Yaskawa INFORM job: neg_x_1.JBI

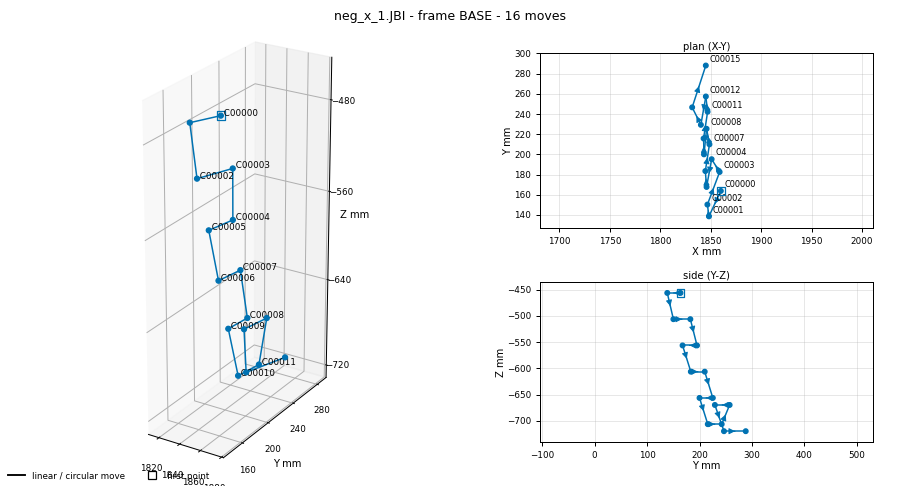
[picture p0: tool path of neg_x_1.JBI in frame BASE, 16 of 18 moves have a stored position in this frame; points joined in program order, loops and branches not executed]
/JOB
//NAME neg_x_1
//POS
///NPOS 16,0,16,0,0,0
///TOOL 0
///POSTYPE BASE
///RECTAN
///RCONF 0,0,0,0,0,0,0,0,0,0,0,0,0,0,0,0,0,0,0,0,0,0,0,0
C00000=1860.009400,163.782870,-456.169200,-175.000000,-80.909620,-24.601701
C00001=1848.219400,138.594450,-456.169200,-175.000000,-80.909620,-24.601701
C00002=1846.699400,150.259350,-506.169200,-175.000000,-80.909620,-24.601701
C00003=1858.829400,182.584150,-506.169200,-175.000000,-80.909620,-24.601701
C00004=1850.899400,195.228650,-556.169200,-175.000000,-80.909620,-24.601701
C00005=1845.879400,167.731640,-556.169200,-175.000000,-80.909620,-24.601701
C00006=1844.649400,183.479050,-606.169200,-175.000000,-80.909620,-24.601701
C00007=1848.749400,209.941950,-606.169200,-175.000000,-80.909620,-24.601701
C00008=1845.889400,225.378650,-656.169200,-175.000000,-80.909620,-24.601701
C00009=1843.319400,200.049150,-656.169200,-175.000000,-80.909620,-24.601701
C00010=1842.919400,215.770950,-706.169200,-175.000000,-80.909620,-24.601701
C00011=1846.899400,242.289250,-706.169200,-175.000000,-80.909620,-24.601701
C00012=1845.159400,257.405150,-669.566660,180.000000,-60.000000,0.000000
C00013=1840.239400,229.288350,-669.566660,180.000000,-60.000000,0.000000
C00014=1831.609400,246.639550,-719.566660,180.000000,-60.000000,0.000000
C00015=1845.119400,288.075850,-719.566660,180.000000,-60.000000,0.000000
///POSTYPE PULSE
///PULSE
EX000=92160
///POSTYPE PULSE
///PULSE
EC00000=92160
EC00001=92160
EC00002=92160
EC00003=92160
EC00004=92160
EC00005=92160
EC00006=92160
EC00007=92160
EC00008=92160
EC00009=92160
EC00010=92160
EC00011=92160
EC00012=92160
EC00013=92160
EC00014=92160
EC00015=92160
//INST
///DATE 2023/08/07 13:53
///ATTR SC,RW,RJ
////FRAME BASE
///GROUP1 RB1,ST1
NOP
MOVJ P009 EX000 VJ=15.00
MOVJ C00000 EC00000 VJ=15.0
CALL JOB:SPYON
MOVL C00001 EC00001 V=150.0
MOVL C00002 EC00002 V=150.0
MOVL C00003 EC00003 V=150.0
MOVL C00004 EC00004 V=150.0
MOVL C00005 EC00005 V=150.0
MOVL C00006 EC00006 V=150.0
MOVL C00007 EC00007 V=150.0
MOVL C00008 EC00008 V=150.0
MOVL C00009 EC00009 V=150.0
MOVL C00010 EC00010 V=150.0
MOVL C00011 EC00011 V=150.0
MOVL C00012 EC00012 V=150.0
MOVL C00013 EC00013 V=150.0
MOVL C00014 EC00014 V=150.0
MOVL C00015 EC00015 V=150.0
CALL JOB:SPYOF
MOVJ P009 VJ=15.00
END
